FUNCTION INTERNAL IncUDINT : UDINT
VAR_INPUT
	refValue		: REFERENCE TO UDINT;
END_VAR

IncUDINT := (refValue := refValue + 1);

END_FUNCTION

(* stored: Version 1.1.0.1, ProductVersion 3.1.4024.0
   POU IncUDINT: Id {82f3f8c5-5683-4bda-9a65-aa0bf43ff118}, SpecialFunc None *)
